ScreenModuleEditorView "valve_ecs8" 1024x768
   SymbolicIOField "mode" at 30,30 size 24x24; TextOn '1'; TextOff '0'; TextList "mode_l"
      Appearance <- "mode"
      ProcessValue <- "mode"
      Visibility <- "mode"
   TextField "x_sig" at 30,9 size 24x24; Text 'X'
      Visibility <- "status_lt"
   TextField "tag" at 17,55 size 115x21; Text 'TAG_NAME_XX'
      Text <- "TAG"
      Visible <- "TAG_VIS"
   Polygon "vlve" at 56,12 size 48x40
      Appearance <- "status_lt"
   IOField "msw_event" at 64,40 size 42x10; FormatPattern FFFFFFFF
      ProcessValue <- "MSW"
      on ObjectChange: "OnObjectChange"
*)

(* ===== HMI "HMI_RT_1" =====
system functions are stored by id; their names below are inferred from use

HMI tags "Default tag table"
   "msw_ext" : UInt, internal
   "msw_status" : UInt, internal
   "mode" : UInt, internal   // 0 -Auto, 2 - Local, 3 -Manual
   "status_lt" : UInt, internal   // 0 -Close; 1 - Open; 2-Moving; 3 - Select; 5 - Fault
   "test" : UInt, internal

text list "mode_l": 0 'A'; 2 'M'; 3 'L'

ScreenModuleEditorView "valve_ecs8" 1024x768
   SymbolicIOField "mode" at 30,30 size 24x24; TextOn '1'; TextOff '0'; TextList "mode_l"
      Appearance <- "mode"
      ProcessValue <- "mode"
      Visibility <- "mode"
   TextField "x_sig" at 30,9 size 24x24; Text 'X'
      Visibility <- "status_lt"
   TextField "tag" at 17,55 size 115x21; Text 'TAG_NAME_XX'
      Text <- "TAG"
      Visible <- "TAG_VIS"
   Polygon "vlve" at 56,16 size 48x32
      Appearance <- "status_lt"
   IOField "msw_event" at 64,40 size 42x10; FormatPattern FFFFFFFF
      ProcessValue <- "MSW"
      on ObjectChange: "OnObjectChange"
*)

(* ===== HMI "HMI_RT_1" =====

text list "mode_l": 0 'A'; 2 'M'; 3 'L'

text list "analog_status": 1 'Normal'; 50 'Activate Block Alarm'; 51 'Activate Advisory Alarm'; 52 'Activate Critical Alarm'; 53 'Unacknowledged Block Alarm'; 54 'Unacknowledged Advisory Alarm'; 55 'Unacknowledged Critical Alarm'; 56 'Init Fail Safe'; 57 'Maintenance Required'; 150 'Open Loop'; 151 'Short Circuit'; 152 'Signal Fault'; 153 'Bad'; 154 'Bad - Configuration Error'; 155 'Bad - Not Connected'; 156 'Bad - Device Failure'; 157 'Bad - No Communication'; 158 'Bad - No Communication'; 159 'Bad - Out of service'; 160 'Bad - Non Measured'; 161 'Bad - Maintenance Alarm'; 162 'Bad - Maintenance Demand'; 163 'Uncertain'; 164 'Uncertain - Last Usable'; 165 'Uncertain - Substiture Set'; 166 'Uncertain - Initial Value'; 167 'Uncertain - Sensor Not Accurate'; 168 'Uncertain - EU range exceeded'; 169 'Uncertain - Sub Normal'; 170 'Uncertain - Configuration Error'; 171 'Simulated Value'; 172 'Calibrating'; 173 'H3 Fatal Alarm'; 174 'L3 Fatal Alarm'; 175 'H2 Alarm'; 176 'L2 Alarm'; 177 'H1 Warning'; 178 'L1 Warning'; 179 'Rate of Change'; 180 'Open Loop'; 181 'Short Circuit'

ScreenModuleEditorView "analog_ecs8" 1024x768
   TextField "tag" at 30,41 size 134x18; Text 'TAG_NAME_XX'
      Text <- "TAG"
      Visible <- "TAG_VIS"
   IOField "I/O field_1" at 64,12 size 100x22; FormatPattern s999999.99
      Appearance <- "MSW.Status"
      FormatPattern <- "FORMAT"
      ProcessValue <- "MSW.VALUE"
      Unit <- "UNIT"
   TextField "output_head_25" at 36,12 size 22x22; Text '!'
      Visibility <- "MSW.EXT"
*)